FUNCTION_BLOCK Temperature EXTENDS SM_Temperature
VAR_INPUT
END_VAR
VAR_OUTPUT
END_VAR
VAR
    _testVar_Temperature : BOOL;
END_VAR

SUPER^();

END_FUNCTION_BLOCK

(* stored: Version 1.1.0.1, ProductVersion 3.1.4018.2
   POU Temperature: Id {5f3a6710-e2e1-44ea-8138-203001a209df}, SpecialFunc None *)
